FUNCTION_BLOCK FB_System_WT_HWW_915
VAR_INPUT
	Freigabe_auto			: BOOL;
	Betrieb_Anford_auto		: BOOL;
	Regelung_Sollw_auto		: REAL;
END_VAR
VAR_OUTPUT
	{attribute 'OPC.UA.DA' := '1'}Steuerung				: ST_System_WT_HWW_Steuerung;		
	{attribute 'OPC.UA.DA' := '1'}Stellwert					: ST_System_WT_HWW_Stellwert;	
	{attribute 'OPC.UA.DA' := '1'}Zustand					: ST_System_WT_HWW_Zustand;		
	{attribute 'OPC.UA.DA' := '1'}Parameter				: ST_System_WT_HWW_Parameter;		
END_VAR
VAR
	Pumpe_215				: FB_PU;
	Pumpe_315				: FB_PU;
	Stellventil_215			: FB_SV;
	Regelventil_215			: FB_RV;	(* 14.07.2020*)
	Stellventil_315			: FB_SV;

	Zustandscheck			: FB_System_WT_HWW_Zustandscheck;
	Logik					: FB_System_WT_HWW_Logik;
	Ablaufsteuerung			: FB_System_WT_HWW_Ablaufsteuerung;
	Sollwertscheck			: FB_System_WT_HWW_Sollwertscheck;
END_VAR
VAR // added by the converter: edge detectors and wires of the graphical bodies
    _w1 : ANY;
END_VAR

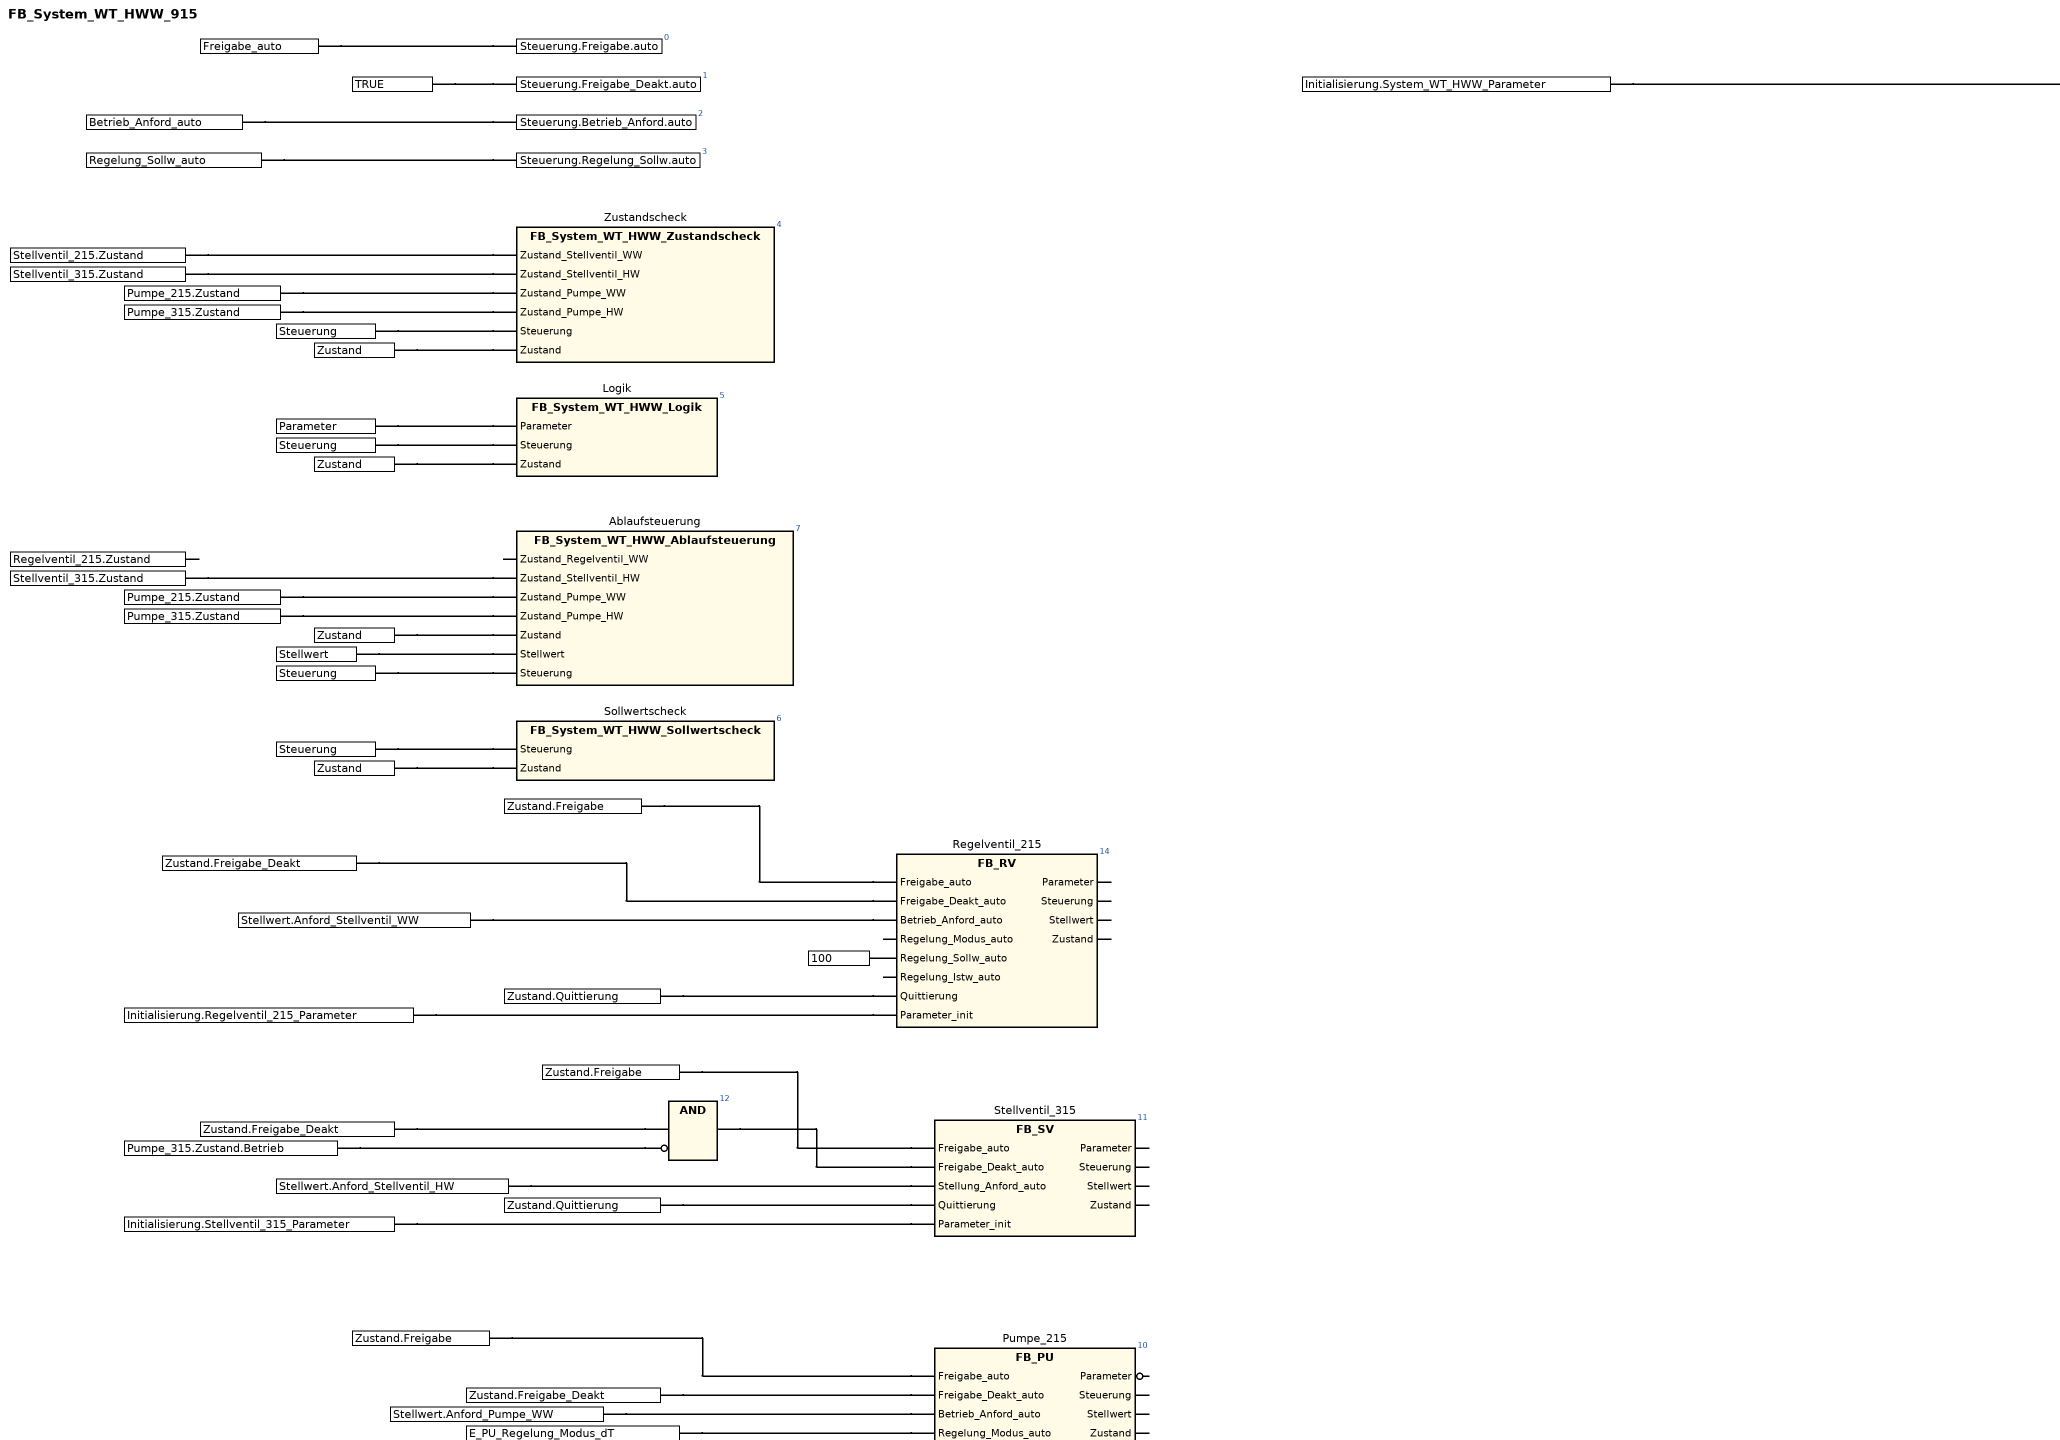
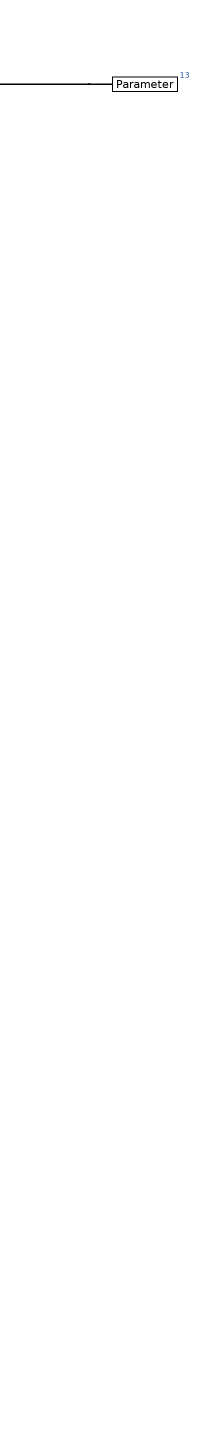
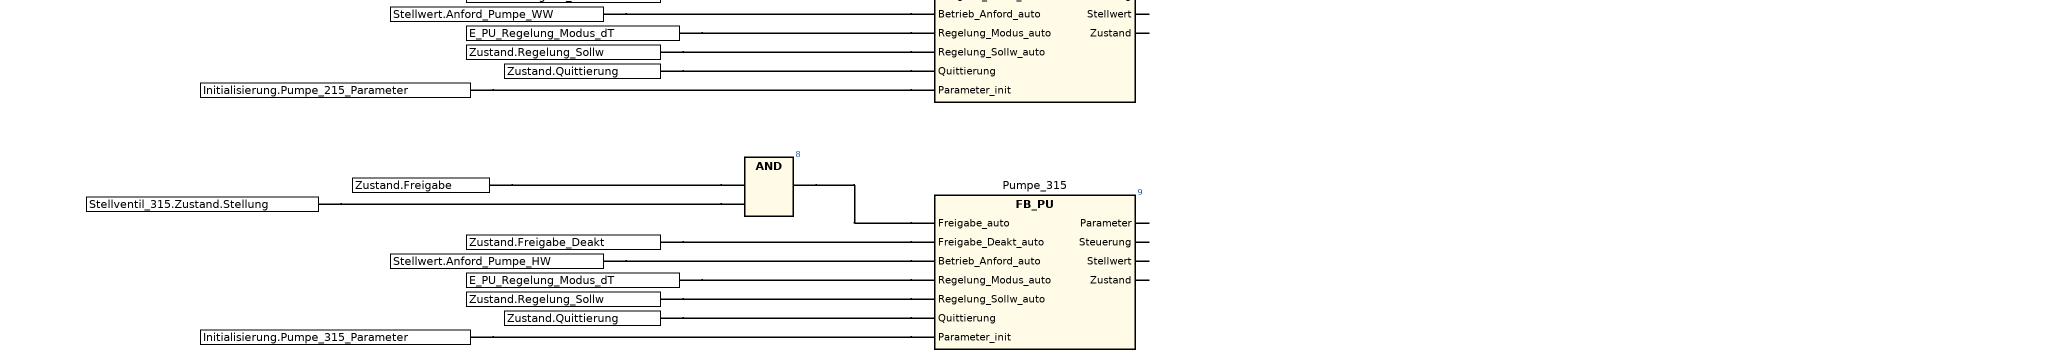
Steuerung.Freigabe.auto := Freigabe_auto;
Steuerung.Freigabe_Deakt.auto := TRUE;
Steuerung.Betrieb_Anford.auto := Betrieb_Anford_auto;
Steuerung.Regelung_Sollw.auto := Regelung_Sollw_auto;
Zustandscheck(
    Zustand_Stellventil_WW := Stellventil_215.Zustand,
    Zustand_Stellventil_HW := Stellventil_315.Zustand,
    Zustand_Pumpe_WW := Pumpe_215.Zustand,
    Zustand_Pumpe_HW := Pumpe_315.Zustand,
    Steuerung := Steuerung,
    Zustand := Zustand); // FB_System_WT_HWW_Zustandscheck
Logik(Parameter := Parameter, Steuerung := Steuerung, Zustand := Zustand); // FB_System_WT_HWW_Logik
Sollwertscheck(Steuerung := Steuerung, Zustand := Zustand); // FB_System_WT_HWW_Sollwertscheck
Ablaufsteuerung(
    Zustand_Stellventil_HW := Stellventil_315.Zustand,
    Zustand_Pumpe_WW := Pumpe_215.Zustand,
    Zustand_Pumpe_HW := Pumpe_315.Zustand,
    Zustand := Zustand,
    Stellwert := Stellwert,
    Steuerung := Steuerung); // FB_System_WT_HWW_Ablaufsteuerung
Pumpe_315(
    Freigabe_auto := Zustand.Freigabe AND Stellventil_315.Zustand.Stellung,
    Freigabe_Deakt_auto := Zustand.Freigabe_Deakt,
    Betrieb_Anford_auto := Stellwert.Anford_Pumpe_HW,
    Regelung_Modus_auto := E_PU_Regelung_Modus_dT,
    Regelung_Sollw_auto := Zustand.Regelung_Sollw,
    Quittierung := Zustand.Quittierung,
    Parameter_init := Initialisierung.Pumpe_315_Parameter); // FB_PU
Pumpe_215(
    Freigabe_auto := Zustand.Freigabe,
    Freigabe_Deakt_auto := Zustand.Freigabe_Deakt,
    Betrieb_Anford_auto := Stellwert.Anford_Pumpe_WW,
    Regelung_Modus_auto := E_PU_Regelung_Modus_dT,
    Regelung_Sollw_auto := Zustand.Regelung_Sollw,
    Quittierung := Zustand.Quittierung,
    Parameter_init := Initialisierung.Pumpe_215_Parameter); // FB_PU
Stellventil_315(
    Freigabe_auto := Zustand.Freigabe,
    Freigabe_Deakt_auto := _w1,
    Stellung_Anford_auto := Stellwert.Anford_Stellventil_HW,
    Quittierung := Zustand.Quittierung,
    Parameter_init := Initialisierung.Stellventil_315_Parameter); // FB_SV
_w1 := Zustand.Freigabe_Deakt AND NOT Pumpe_315.Zustand.Betrieb;
Parameter := Initialisierung.System_WT_HWW_Parameter;
Regelventil_215(
    Freigabe_auto := Zustand.Freigabe,
    Freigabe_Deakt_auto := Zustand.Freigabe_Deakt,
    Betrieb_Anford_auto := Stellwert.Anford_Stellventil_WW,
    Regelung_Sollw_auto := 100,
    Quittierung := Zustand.Quittierung,
    Parameter_init := Initialisierung.Regelventil_215_Parameter); // FB_RV
// Regelventil_215.Zustand: input not connected

END_FUNCTION_BLOCK

(* stored: Version 1.1.0.1, ProductVersion 3.1.4024.9
   POU FB_System_WT_HWW_915: Id {6de39ffa-026d-429a-bf4c-1a3860737e53}, SpecialFunc None *)
